KUKA KRL data list: kuka_eki_hw_interface.dat

       &ACCESS RVP
&REL 25
&PARAM DISKPATH = Program
DEFDAT  kuka_eki_hw_int_eje_ext
EXT  bas (BAS_COMMAND  :IN,REAL  :IN )
DECL BASIS_SUGG_T LAST_BASIS={POINT1[] "P3                      ",POINT2[] "P3                      ",CP_PARAMS[] "CPDAT0                  ",PTP_PARAMS[] "PDAT3                   ",CONT[] "                        ",CP_VEL[] "2.0                     ",PTP_VEL[] "100                     ",SYNC_PARAMS[] "SYNCDAT                 ",SPL_NAME[] "S0                      ",A_PARAMS[] "ADAT0                   "}
DECL E6POS XP1={X 610.705627,Y 0.334120929,Z 1934.93970,A 176.606598,B 89.6755600,C 176.570938,S 18,T 3,E1 0.00137973239,E2 -0.00409854297,E3 0.0,E4 0.0,E5 0.0,E6 0.0}
DECL FDAT FP1={TOOL_NO 1,BASE_NO 0,IPO_FRAME #BASE,POINT2[] " ",TQ_STATE FALSE}
DECL PDAT PPDAT1={VEL 100.000,ACC 100.000,APO_DIST 100.000,GEAR_JERK 50.0000,EXAX_IGN 0}
DECL E6POS XP2={X 605.194580,Y 0.321840733,Z 1938.04089,A 137.126724,B 89.9518280,C 137.090195,S 18,T 11,E1 -4.60337210,E2 0.153725460,E3 0.0,E4 0.0,E5 0.0,E6 0.0}
DECL FDAT FP2={TOOL_NO 1,BASE_NO 0,IPO_FRAME #BASE,POINT2[] " ",TQ_STATE FALSE}
DECL PDAT PPDAT2={VEL 100.000,ACC 100.000,APO_DIST 100.000,GEAR_JERK 50.0000,EXAX_IGN 0}
DECL E6POS XP3={X 605.196411,Y 0.321772158,Z 1938.04285,A 136.397385,B 89.9510727,C 136.360870,S 18,T 34,E1 3.16293621,E2 -5.24398518,E3 0.0,E4 0.0,E5 0.0,E6 0.0}
DECL FDAT FP3={TOOL_NO 1,BASE_NO 0,IPO_FRAME #BASE,POINT2[] " ",TQ_STATE FALSE}
DECL PDAT PPDAT3={VEL 100.000,ACC 100.000,APO_DIST 100.000,GEAR_JERK 50.0000,EXAX_IGN 0}
ENDDAT
